FUNCTION_BLOCK FB_Drive IMPLEMENTS I_Drive
VAR_IN_OUT
    Axis : AXIS_REF; 
END_VAR

VAR_INPUT
    // --- External Commands ---
    bEnableCmd  : BOOL; 
END_VAR

VAR
    // --- Standard PLCopen Motion Blocks ---
    fbPower     : MC_Power;
    fbReset     : MC_Reset;
    fbStop      : MC_Stop;
    fbMoveAbs   : MC_MoveAbsolute;
    fbMoveVel   : MC_MoveVelocity;
    fbHome      : MC_Home;
END_VAR

// 1. Always Update the Axis Status
Axis.ReadStatus();

// 2. Power Control (Torque on/off)
fbPower(
    Axis := Axis,
    Enable := bEnableCmd,
    Enable_Positive := bEnableCmd,
    Enable_Negative := bEnableCmd
);

// 3. Call the Motion Function Blocks
// Note: We call them here so they can process their internal state machines
fbReset(Axis := Axis);
fbStop(Axis := Axis);
fbMoveAbs(Axis := Axis);
fbMoveVel(Axis := Axis);
fbHome(Axis := Axis);

// =========================================================
// CORRECTED TRIGGER RESET LOGIC
// =========================================================
// The Execute signals are now only dropped once the NC block 
// finishes its operation. This ensures the FB state machines 
// complete their execution and accurately reflect P_Busy.

IF fbReset.Done OR fbReset.Error THEN
    fbReset.Execute := FALSE;
END_IF

IF fbStop.Done OR fbStop.CommandAborted OR fbStop.Error THEN
    fbStop.Execute := FALSE;
END_IF

IF fbMoveAbs.Done OR fbMoveAbs.CommandAborted OR fbMoveAbs.Error THEN
    fbMoveAbs.Execute := FALSE;
END_IF

// ---> FIX: Now includes fbMoveVel.InVelocity to unlock the master profile
IF fbMoveVel.InVelocity OR fbMoveVel.CommandAborted OR fbMoveVel.Error THEN
    fbMoveVel.Execute := FALSE;
END_IF

IF fbHome.Done OR fbHome.CommandAborted OR fbHome.Error THEN
    fbHome.Execute := FALSE;
END_IF

METHOD M_Home : BOOL
// Trigger a rising edge on the internal home block
// Note: We use the default homing mode configured in the TwinCAT NC Axis
fbHome.bCalibrationCam := FALSE; 
fbHome.Execute := TRUE;

M_Home := TRUE;
END_METHOD

METHOD M_MoveAbs : BOOL
VAR_INPUT
	(* Target position in mm or degrees*)
	fPosition	: LREAL;
	(* Speed for this move*)
	fVelocity	: LREAL;
END_VAR
// Trigger a rising edge on the internal motion block
fbMoveAbs.Position := fPosition;
fbMoveAbs.Velocity := fVelocity;
fbMoveAbs.Execute := TRUE; 

M_MoveAbs := TRUE; // Return TRUE to show the command was received
END_METHOD

METHOD M_MoveVelocity : BOOL
VAR_INPUT
    fVelocity   : LREAL;         // Target speed in mm/s
    nDirection  : MC_Direction;  // 1 = Positive, 2 = Negative, 3 = Current
END_VAR
// Pass the inputs to the underlying PLCopen block
fbMoveVel.Velocity  := fVelocity;
fbMoveVel.Direction := nDirection;
fbMoveVel.Execute   := TRUE;

M_MoveVelocity := TRUE;
END_METHOD

METHOD M_Reset : BOOL
fbReset.Execute := TRUE; M_Reset := TRUE;
END_METHOD

METHOD M_Stop : BOOL
fbStop.Execute := TRUE; M_Stop := TRUE;
END_METHOD

PROPERTY P_Axis : REFERENCE TO AXIS_REF
GET
P_Axis REF= Axis; // This creates a 'link' to the real Axis variable
END_GET
END_PROPERTY

PROPERTY P_Busy : BOOL
GET
// The axis is busy if it is physically moving or if a move block is still active
P_Busy := Axis.Status.Moving OR fbMoveAbs.Busy OR fbMoveVel.Busy OR fbHome.Busy;
END_GET
END_PROPERTY

PROPERTY P_Enabled : BOOL
GET
P_Enabled := bEnableCmd;
END_GET
SET
bEnableCmd := P_Enabled;
END_SET
END_PROPERTY

PROPERTY P_Error : BOOL
GET
P_Error := Axis.Status.Error;
END_GET
END_PROPERTY

PROPERTY P_Ready : BOOL
GET
P_Ready := Axis.Status.Operational;
END_GET
END_PROPERTY

END_FUNCTION_BLOCK

(* stored: Version 1.1.0.1
   POU FB_Drive: Id {29575593-8274-429c-a355-871bac34c303}, SpecialFunc None
   Method M_Home: Id {7790ed11-5148-4807-a00e-287e41768cda}
   Method M_MoveAbs: Id {91be8eab-f779-49c3-9c91-e8161a59ed82}
   Method M_MoveVelocity: Id {37e662dd-1514-4118-a818-f288d90d7c84}
   Method M_Reset: Id {b7138b05-71aa-42a5-bcb7-54cd0cd5d5d0}
   Method M_Stop: Id {a8aa22d7-69f3-4b58-8bbe-8959b5116ba7}
   Property P_Axis: Id {c438ebb6-f4fa-4896-b4fc-45b79fc5096e}
   Get Get: Id {971a64fc-7619-44e1-b200-2ade4597c9b2}
   Property P_Busy: Id {0954bfd9-2a2f-442b-88a7-0fc7aa654616}
   Get Get: Id {af39002d-3e39-450d-9298-2d3614d5dde1}
   Property P_Enabled: Id {aa86077e-a730-425c-9d71-e45f00711c2b}
   Get Get: Id {92730983-4549-44bf-8946-dcdf46ccfe10}
   Set Set: Id {a6e6e813-1d0d-42b7-b058-ad03723ae751}
   Property P_Error: Id {dc88c766-3499-41ab-b41f-3c6f5290d649}
   Get Get: Id {a36b31b8-1fee-448b-b160-4c3cf7dd54df}
   Property P_Ready: Id {614d4749-6d6c-42bf-a79f-dfd89216bbcd}
   Get Get: Id {9697a46b-6c06-4d27-8b82-b857d1608699} *)
